FUNCTION_BLOCK ThreeConCtl (* Composite Function Block Type *)
  (* Standard: 61499-2 *)
  (* Version 0.2, 2003-12-05, JHC, Rockwell Automation, Renamed from NEWCOMPFB. *)
  (* Version 0.1, 2002-01-08, JHC, Rockwell Automation, Added DLY FB as example. *)
  (* Version 0.0, 2000-05-27, JHC, Rockwell Automation *)
  (* Compiler header: package fb.rt.cs725; *)
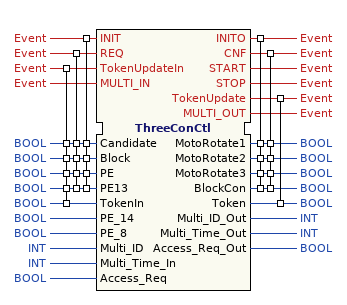
  EVENT_INPUT
    INIT WITH Candidate, Block, PE, PE13; (* Initialization Request *)
    REQ WITH Block, Candidate, PE, PE13; (* Normal Execution Request *)
    TokenUpdateIn WITH Candidate, Block, PE, PE13, TokenIn;
    MULTI_IN;
  END_EVENT
  EVENT_OUTPUT
    INITO WITH MotoRotate1, MotoRotate2, MotoRotate3, BlockCon; (* Initialization Confirm *)
    CNF WITH MotoRotate1, MotoRotate2, MotoRotate3, BlockCon; (* Execution Confirmation *)
    START;
    STOP;
    TokenUpdate WITH Token;
    MULTI_OUT;
  END_EVENT
  VAR_INPUT
    Candidate : BOOL;
    Block : BOOL;
    PE : BOOL;
    PE13 : BOOL;
    TokenIn : BOOL;
    PE_14 : BOOL;
    PE_8 : BOOL;
    Multi_ID : INT;
    Multi_Time_In : INT;
    Access_Req : BOOL;
  END_VAR
  VAR_OUTPUT
    MotoRotate1 : BOOL;
    MotoRotate2 : BOOL;
    MotoRotate3 : BOOL;
    BlockCon : BOOL;
    Token : BOOL;
    Multi_ID_Out : INT;
    Multi_Time_Out : INT;
    Access_Req_Out : BOOL;
  END_VAR
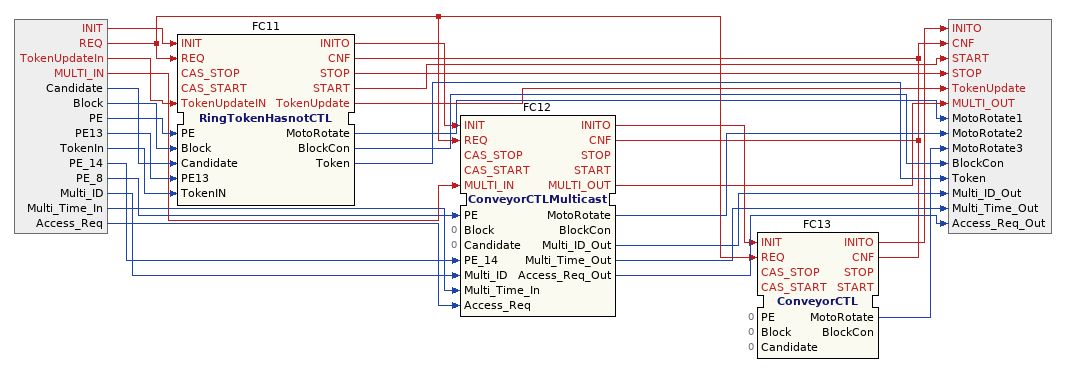
  FBS
    FC11 : RingTokenHasnotCTL;
    FC12 : ConveyorCTLMulticast(Block := 0, Candidate := 0);
    FC13 : ConveyorCTL(PE := 0, Block := 0, Candidate := 0);
  END_FBS
  EVENT_CONNECTIONS
    INIT TO FC11.INIT;
    REQ TO FC11.REQ;
    FC11.INITO TO FC12.INIT;
    FC12.INITO TO FC13.INIT;
    FC13.INITO TO INITO;
    FC13.CNF TO CNF;
    FC11.STOP TO STOP;
    FC11.START TO START;
    REQ TO FC12.REQ;
    REQ TO FC13.REQ;
    FC11.CNF TO CNF;
    FC12.CNF TO CNF;
    TokenUpdateIn TO FC11.TokenUpdateIN;
    FC11.TokenUpdate TO TokenUpdate;
    MULTI_IN TO FC12.MULTI_IN;
    FC12.MULTI_OUT TO MULTI_OUT;
  END_CONNECTIONS
  DATA_CONNECTIONS
    FC13.MotoRotate TO MotoRotate3;
    FC12.MotoRotate TO MotoRotate2;
    FC11.MotoRotate TO MotoRotate1;
    PE TO FC11.PE;
    Block TO FC11.Block;
    FC11.BlockCon TO BlockCon;
    Candidate TO FC11.Candidate;
    PE13 TO FC11.PE13;
    TokenIn TO FC11.TokenIN;
    FC11.Token TO Token;
    PE_8 TO FC12.PE;
    FC12.Multi_ID_Out TO Multi_ID_Out;
    FC12.Multi_Time_Out TO Multi_Time_Out;
    FC12.Access_Req_Out TO Access_Req_Out;
    PE_14 TO FC12.PE_14;
    Multi_ID TO FC12.Multi_ID;
    Multi_Time_In TO FC12.Multi_Time_In;
    Access_Req TO FC12.Access_Req;
  END_CONNECTIONS
END_FUNCTION_BLOCK
